{library PRIVATE}
(*
  Private Funtcion:
  To get an Instance status.
*)
FUNCTION _GetInstance : INSTANCE_STATUS
VAR_INPUT
	Instance:			INT;				(* Instance, a number concatenated by SationNumber (1-INSTANCE_MAX_NUMBER_OF_STATIONS) and DeviceNumber (1-INSTANCE_MAX_NUMBER_OF_DEVICES). Instance is defined as: StaionNumber*100+DeviceNumber *)
END_VAR
VAR
	StationDevice: 	INT;
	StationNumber: 	INT;
END_VAR

_GetInstance:=INSTANCE_STATUS.INSTANCE_STATUS_UNKNOWN;

IF _CheckInstance(Instance) THEN
	StationNumber:=Instance/100;
	StationDevice:=Instance-StationNumber*100;
	_GetInstance:=ComGVL._Instance[StationNumber, StationDevice];
END_IF;

END_FUNCTION

(* stored: Version 1.1.0.1, ProductVersion 3.1.4024.2
   POU _GetInstance: Id {281c7209-503e-4041-a663-f24202d9a9e5}, SpecialFunc None *)
